PROGRAM prgTestAuxsFuns
VAR
	blink:FB_Blink;
	rBlinkOn:LREAL:=0.5;
	rBlinkOff:LREAL:=0.3;
	bOutputBlink: BOOL;
END_VAR

blink(tON:= LREAL_TO_TIME(rBlinkOn*1000), tOff:=LREAL_TO_TIME(rBlinkOff*1000) , output=> bOutputBlink);

END_PROGRAM

(* stored: Version 1.1.0.1, ProductVersion 3.1.4024.12
   POU prgTestAuxsFuns: Id {ec954905-60b3-4502-9520-151971f6a1fe}, SpecialFunc None *)
